PROGRAM MAIN
VAR
	ton_a 	: TON := (PT:=T#1S);
	ton_b	: TON := (PT:=T#0.1S);
	n_cnt_a : UINT := 1;  // 1/s
	n_cnt_b : UINT := 2; // 1/100ms
	n_cnt_c : UINT := 3; // 1/ms
END_VAR

ton_a(IN:= NOT ton_a.Q);
ton_b(IN:= NOT ton_b.Q);

IF ton_a.Q THEN
	n_cnt_a := n_cnt_a + 1;
END_IF

IF ton_b.Q THEN
	n_cnt_b := n_cnt_b + 1;
END_IF

n_cnt_c := n_cnt_c + 1;

END_PROGRAM

(* stored: Version 1.1.0.1, ProductVersion 3.1.4024.11
   POU MAIN: Id {28f7ac37-e2b1-4a38-ba81-9cc3a31bdfdf}, SpecialFunc None *)
